PROGRAM MAIN
VAR
END_VAR

END_PROGRAM

(* stored: Version 1.1.0.1
   POU MAIN: Id {0d04f596-3b55-45ee-a755-3c84db3b4cc3} *)
